SUBAPPLICATION mapping_NumericValue (* Subapplication Type *)
  (* Standard: 61499-2 *)
  (* Version 1.0, 2023-01-29, Franz *)
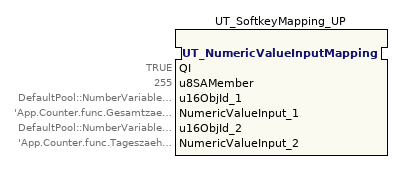
  FBS
    UT_SoftkeyMapping_UP : UT_NumericValueInputMapping(QI := TRUE, u8SAMember := 255, u16ObjId_1 := DefaultPool::NumberVariable_Gesamtziel, NumericValueInput_1 := 'App.Counter.func.GesamtzaehlerVergleich.IN_NumberVariable', u16ObjId_2 := DefaultPool::NumberVariable_Tagesziel, NumericValueInput_2 := 'App.Counter.func.TageszaehlerVergleich.IN_NumberVariable');
  END_FBS
END_SUBAPPLICATION
